INTERFACE IBasicElement

METHOD GetModelState
VAR_INPUT
END_VAR
VAR_OUTPUT
    xDone : BOOL;
    xBusy : BOOL;
    xError : BOOL;
    xAborted : BOOL;
    iErrorID : UDINT;
	UniqueErrorCode : STRING;
END_VAR
END_METHOD

METHOD GetName : STRING
VAR_INPUT
END_VAR
END_METHOD

END_INTERFACE

(* stored: Version 1.1.0.1, ProductVersion 3.1.4024.13
   Itf IBasicElement: Id {26d4507e-e06d-4253-9642-41e206344b1d}
   Method GetModelState: Id {f7b30fda-c760-4669-af64-dc3fa3d6ad6e}
   Method GetName: Id {baf1da5f-3fb9-43d4-a21d-161c0b854311} *)
